TYPE OutputBase_10CEE7DE :
STRUCT
END_STRUCT
END_TYPE

(* stored: Version 1.2.0.0, ProductVersion 3.1.4024.9
   DUT OutputBase_10CEE7DE: Id {fceadb77-2956-4391-a611-56ccc996705e} *)
